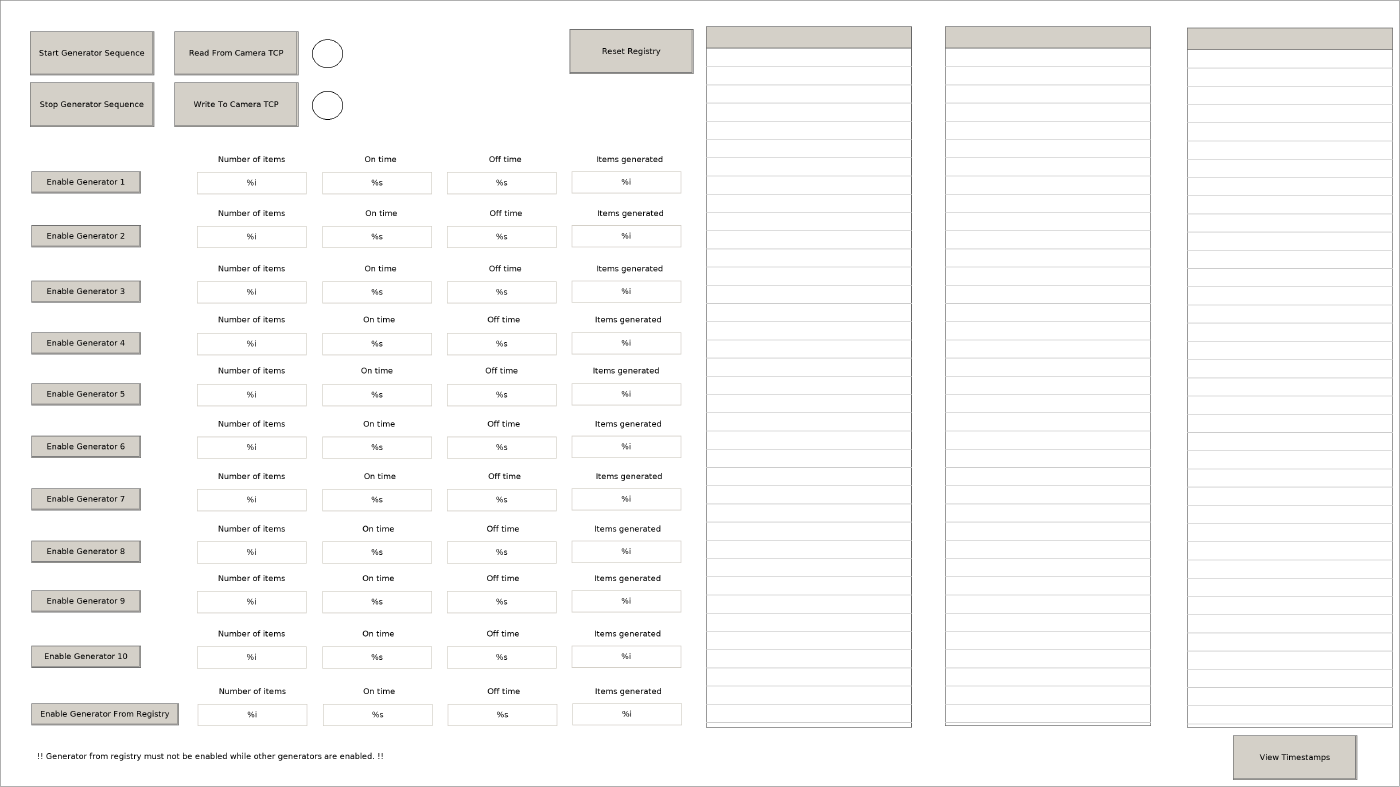
VISUALIZATION ItemSimulator  // 1920x1080
    Button (43,235 150x30), "Enable Generator 1", colour toggle: PRG_Simulator.stItemGen1.bEnableGenerator
        toggle PRG_Simulator.stItemGen1.bEnableGenerator
    Textfield (270,236 150x30), "%i", text variable: PRG_Simulator.stItemGen1.nNumberOfPulses
        OnMouseClick: write the text variable via Default
    Textfield (442,236 150x30), "%s", text variable: PRG_Simulator.stItemGen1.tTimeOnPulse, text index: PRG_Simulator.stItemGen1.tTimeOnPulse
        OnMouseClick: write the text variable via Default
    Textfield (613,236 150x30), "%s", text variable: PRG_Simulator.stItemGen1.tTimeOffPulse, text index: PRG_Simulator.stItemGen1.tTimeOffPulse
        OnMouseClick: write the text variable via Default
    Label (270,204 150x30), "Number of items"
    Label (447,204 150x30), "On time"
    Label (618,204 150x30), "Off time"
    Textfield (784,235 150x30), "%i", text variable: PRG_Simulator.fbItemGenerator.fbItemGen1.uiCount, input disabled if: TRUE, text index: PRG_Simulator.stItemGen1.nNumberOfPulses
        OnMouseClick: write the text variable via Default
    Label (789,204 150x30), "Items generated"
    Button (41,43 170x60), "Start Generator Sequence"
        OnMouseDown: execute { PRG_Simulator.bStartGenerator := TRUE; }
    Button (41,113 170x61), "Stop Generator Sequence"
        OnMouseDown: execute { PRG_Simulator.bStopGenerator := TRUE; }
    Button (43,309 150x30), "Enable Generator 2", colour toggle: PRG_Simulator.stItemGen2.bEnableGenerator
        toggle PRG_Simulator.stItemGen2.bEnableGenerator
    Textfield (270,310 150x30), "%i", text variable: PRG_Simulator.stItemGen2.nNumberOfPulses
        OnMouseClick: write the text variable via Default
    Textfield (442,310 150x30), "%s", text variable: PRG_Simulator.stItemGen2.tTimeOnPulse
        OnMouseClick: write the text variable via Default
    Textfield (613,310 150x30), "%s", text variable: PRG_Simulator.stItemGen2.tTimeOffPulse
        OnMouseClick: write the text variable via Default
    Label (270,278 150x30), "Number of items"
    Label (448,278 150x30), "On time"
    Label (619,278 150x30), "Off time"
    Textfield (784,309 150x30), "%i", text variable: PRG_Simulator.fbItemGenerator.fbItemGen2.uiCount, input disabled if: TRUE
        OnMouseClick: write the text variable via Default
    Label (790,278 150x30), "Items generated"
    Button (43,385 150x30), "Enable Generator 3", colour toggle: PRG_Simulator.stItemGen3.bEnableGenerator
        toggle PRG_Simulator.stItemGen3.bEnableGenerator
    Textfield (270,386 150x30), "%i", text variable: PRG_Simulator.stItemGen3.nNumberOfPulses
        OnMouseClick: write the text variable via Default
    Textfield (442,386 150x30), "%s", text variable: PRG_Simulator.stItemGen3.tTimeOnPulse
        OnMouseClick: write the text variable via Default
    Textfield (613,386 150x30), "%s", text variable: PRG_Simulator.stItemGen3.tTimeOffPulse
        OnMouseClick: write the text variable via Default
    Label (270,354 150x30), "Number of items"
    Label (447,354 150x30), "On time"
    Label (618,354 150x30), "Off time"
    Textfield (784,385 150x30), "%i", text variable: PRG_Simulator.fbItemGenerator.fbItemGen3.uiCount, input disabled if: TRUE
        OnMouseClick: write the text variable via Default
    Label (789,354 150x30), "Items generated"
    Button (43,456 150x30), "Enable Generator 4", colour toggle: PRG_Simulator.stItemGen4.bEnableGenerator
        toggle PRG_Simulator.stItemGen4.bEnableGenerator
    Textfield (270,457 150x30), "%i", text variable: PRG_Simulator.stItemGen4.nNumberOfPulses
        OnMouseClick: write the text variable via Default
    Textfield (442,457 150x30), "%s", text variable: PRG_Simulator.stItemGen4.tTimeOnPulse
        OnMouseClick: write the text variable via Default
    Textfield (613,457 150x30), "%s", text variable: PRG_Simulator.stItemGen4.tTimeOffPulse
        OnMouseClick: write the text variable via Default
    Label (270,424 150x30), "Number of items"
    Label (445,424 150x30), "On time"
    Label (616,424 150x30), "Off time"
    Textfield (784,456 150x30), "%i", text variable: PRG_Simulator.fbItemGenerator.fbItemGen4.uiCount, input disabled if: TRUE
        OnMouseClick: write the text variable via Default
    Label (787,424 150x30), "Items generated"
    Button (43,526 150x30), "Enable Generator 5", colour toggle: PRG_Simulator.stItemGen5.bEnableGenerator
        toggle PRG_Simulator.stItemGen5.bEnableGenerator
    Textfield (270,527 150x30), "%i", text variable: PRG_Simulator.stItemGen5.nNumberOfPulses
        OnMouseClick: write the text variable via Default
    Textfield (442,527 150x30), "%s", text variable: PRG_Simulator.stItemGen5.tTimeOnPulse
        OnMouseClick: write the text variable via Default
    Textfield (613,527 150x30), "%s", text variable: PRG_Simulator.stItemGen5.tTimeOffPulse
        OnMouseClick: write the text variable via Default
    Label (270,494 150x30), "Number of items"
    Label (442,494 150x30), "On time"
    Label (613,494 150x30), "Off time"
    Textfield (784,526 150x30), "%i", text variable: PRG_Simulator.fbItemGenerator.fbItemGen5.uiCount, input disabled if: TRUE
        OnMouseClick: write the text variable via Default
    Label (784,494 150x30), "Items generated"
    Button (43,598 150x30), "Enable Generator 6", colour toggle: PRG_Simulator.stItemGen6.bEnableGenerator
        toggle PRG_Simulator.stItemGen6.bEnableGenerator
    Textfield (270,599 150x30), "%i", text variable: PRG_Simulator.stItemGen6.nNumberOfPulses
        OnMouseClick: write the text variable via Default
    Textfield (442,599 150x30), "%s", text variable: PRG_Simulator.stItemGen6.tTimeOnPulse
        OnMouseClick: write the text variable via Default
    Textfield (613,599 150x30), "%s", text variable: PRG_Simulator.stItemGen6.tTimeOffPulse
        OnMouseClick: write the text variable via Default
    Label (270,567 150x30), "Number of items"
    Label (445,567 150x30), "On time"
    Label (616,567 150x30), "Off time"
    Textfield (784,598 150x30), "%i", text variable: PRG_Simulator.fbItemGenerator.fbItemGen6.uiCount, input disabled if: TRUE
        OnMouseClick: write the text variable via Default
    Label (787,567 150x30), "Items generated"
    Button (43,670 150x30), "Enable Generator 7", colour toggle: PRG_Simulator.stItemGen7.bEnableGenerator
        toggle PRG_Simulator.stItemGen7.bEnableGenerator
    Textfield (270,671 150x30), "%i", text variable: PRG_Simulator.stItemGen7.nNumberOfPulses
        OnMouseClick: write the text variable via Default
    Textfield (442,671 150x30), "%s", text variable: PRG_Simulator.stItemGen7.tTimeOnPulse
        OnMouseClick: write the text variable via Default
    Textfield (613,671 150x30), "%s", text variable: PRG_Simulator.stItemGen7.tTimeOffPulse
        OnMouseClick: write the text variable via Default
    Label (270,639 150x30), "Number of items"
    Label (446,639 150x30), "On time"
    Label (617,639 150x30), "Off time"
    Textfield (784,670 150x30), "%i", text variable: PRG_Simulator.fbItemGenerator.fbItemGen7.uiCount, input disabled if: TRUE
        OnMouseClick: write the text variable via Default
    Label (788,639 150x30), "Items generated"
    Button (43,742 150x30), "Enable Generator 8", colour toggle: PRG_Simulator.stItemGen8.bEnableGenerator
        toggle PRG_Simulator.stItemGen8.bEnableGenerator
    Textfield (270,743 150x30), "%i", text variable: PRG_Simulator.stItemGen8.nNumberOfPulses
        OnMouseClick: write the text variable via Default
    Textfield (442,743 150x30), "%s", text variable: PRG_Simulator.stItemGen8.tTimeOnPulse
        OnMouseClick: write the text variable via Default
    Textfield (613,743 150x30), "%s", text variable: PRG_Simulator.stItemGen8.tTimeOffPulse
        OnMouseClick: write the text variable via Default
    Label (270,711 150x30), "Number of items"
    Label (444,711 150x30), "On time"
    Label (615,711 150x30), "Off time"
    Textfield (784,742 150x30), "%i", text variable: PRG_Simulator.fbItemGenerator.fbItemGen8.uiCount, input disabled if: TRUE
        OnMouseClick: write the text variable via Default
    Label (786,711 150x30), "Items generated"
    Button (43,810 150x30), "Enable Generator 9", colour toggle: PRG_Simulator.stItemGen9.bEnableGenerator
        toggle PRG_Simulator.stItemGen9.bEnableGenerator
    Textfield (270,811 150x30), "%i", text variable: PRG_Simulator.stItemGen9.nNumberOfPulses
        OnMouseClick: write the text variable via Default
    Textfield (442,811 150x30), "%s", text variable: PRG_Simulator.stItemGen9.tTimeOnPulse
        OnMouseClick: write the text variable via Default
    Textfield (613,811 150x30), "%s", text variable: PRG_Simulator.stItemGen9.tTimeOffPulse
        OnMouseClick: write the text variable via Default
    Label (270,779 150x30), "Number of items"
    Label (444,779 150x30), "On time"
    Label (615,779 150x30), "Off time"
    Textfield (784,810 150x30), "%i", text variable: PRG_Simulator.fbItemGenerator.fbItemGen9.uiCount, input disabled if: TRUE
        OnMouseClick: write the text variable via Default
    Label (786,779 150x30), "Items generated"
    Button (43,886 150x30), "Enable Generator 10", colour toggle: PRG_Simulator.stItemGen10.bEnableGenerator
        toggle PRG_Simulator.stItemGen10.bEnableGenerator
    Textfield (270,887 150x30), "%i", text variable: PRG_Simulator.stItemGen10.nNumberOfPulses
        OnMouseClick: write the text variable via Default
    Textfield (442,887 150x30), "%s", text variable: PRG_Simulator.stItemGen10.tTimeOnPulse
        OnMouseClick: write the text variable via Default
    Textfield (613,887 150x30), "%s", text variable: PRG_Simulator.stItemGen10.tTimeOffPulse
        OnMouseClick: write the text variable via Default
    Label (270,855 150x30), "Number of items"
    Label (444,855 150x30), "On time"
    Label (615,855 150x30), "Off time"
    Textfield (784,886 150x30), "%i", text variable: PRG_Simulator.fbItemGenerator.fbItemGen10.uiCount, input disabled if: TRUE
        OnMouseClick: write the text variable via Default
    Label (786,855 150x30), "Items generated"
    Textfield (271,966 150x30), "%i", text variable: PRG_Simulator.stItemGenFromReg.nNumberOfPulses, input disabled if: TRUE
        OnMouseClick: write the text variable via Default
    Textfield (443,966 150x30), "%s", text variable: PRG_Simulator.stItemGenFromReg.tTimeOnPulse, input disabled if: TRUE
        OnMouseClick: write the text variable via Default
    Textfield (614,966 150x30), "%s", text variable: PRG_Simulator.stItemGenFromReg.tTimeOffPulse, input disabled if: TRUE
        OnMouseClick: write the text variable via Default
    Label (271,934 150x30), "Number of items"
    Label (445,934 150x30), "On time"
    Label (616,934 150x30), "Off time"
    Textfield (785,965 150x30), "%i", text variable: PRG_Simulator.fbItemGenerator.fbItemGenFromReg.uiCount, input disabled if: TRUE
        OnMouseClick: write the text variable via Default
    Label (787,934 150x30), "Items generated"
    Button (43,965 202x30), "Enable Generator From Registry", colour toggle: PRG_Simulator.stItemGenFromReg.bEnableGenerator
        toggle PRG_Simulator.stItemGenFromReg.bEnableGenerator
    Table (968,36 282x962), data array: PRG_Simulator.aItemOnTimeRegistry
        p3854506369: PRG_Simulator.aItemOnTimeRegistry[INDEX]
        p2232123230: On time From Registry
    Table (1296,36 282x960), data array: PRG_Simulator.aItemOffTimeRegistry
        p3854506369: PRG_Simulator.aItemOffTimeRegistry[INDEX]
        p2232123230: Off Time From Registry
    Button (781,40 170x61), "Reset Registry"
        toggle GVL_ItemSimulator.bResetRegistry
    Label (20,1023 537x30), "!! Generator from registry must not be enabled while other generators are enabled. !!"
    Table (1628,38 282x960), data array: PRG_TCPIP.aItemEANRegistry
        p3854506369: PRG_TCPIP.aItemEANRegistry[INDEX]
        p2232123230: EAN String From Registry
    Button (239,43 170x60), "Read From Camera TCP"
        OnMouseDown: execute { PRG_TCPIP.bConnectCameraRead := TRUE; }
    Button (239,113 170x61), "Write To Camera TCP"
        OnMouseDown: execute { PRG_TCPIP.bConnectCameraWrite := TRUE; }
    Button (1691,1009 170x61), "View Timestamps"
        OnMouseClick: change screen: TimeStampOnItems
    Ellipse (428,54 42x39), colour toggle: PRG_TCPIP.bConnectedCameraRead, colour variable: 16#FFFFFFFF
        p2167032090: 16#FF78CE22
    Ellipse (428,125 42x39), colour toggle: PRG_TCPIP.bConnectedCameraWrite, colour variable: 16#FFFFFFFF
        p2167032090: 16#FF78CE22
END_VISUALIZATION

(* stored: Version 1.1.0.1, ProductVersion 3.1.4024.12
   Visu ItemSimulator: Id {0fccc92e-fff4-4187-a53b-4c3eb227158a} *)
